(* IEC 61131-3 sources: ATCMcontrol_Engineering/src/TargetBase/Libs/ATCM_IEC1131_3/table_22, 158 files *)

(* ---- bool_to_byte.st ---- *)
(*[[
    UserURL= "ATCMfile:BOOL_TO_BYTE.htm"
]]*)

FUNCTION BOOL_TO_BYTE : BYTE
VAR_INPUT
    IN : BOOL;
END_VAR

inline { VMOP(bool_to_byte) }

END_FUNCTION

(* ---- bool_to_dint.st ---- *)
(*[[
    UserURL= "ATCMfile:BOOL_TO_DINT.htm"
]]*)

FUNCTION BOOL_TO_DINT : DINT
VAR_INPUT
    IN : BOOL;
END_VAR

inline{ VMOP(bool_to_dword) }

END_FUNCTION

(* ---- bool_to_dword.st ---- *)
(*[[
    UserURL= "ATCMfile:BOOL_TO_DWORD.htm"
]]*)

FUNCTION BOOL_TO_DWORD : DWORD
VAR_INPUT
    IN : BOOL;
END_VAR

inline{ VMOP(bool_to_dword) }

END_FUNCTION

(* ---- bool_to_int.st ---- *)
(*[[
    UserURL= "ATCMfile:BOOL_TO_DINT.htm"
]]*)

FUNCTION BOOL_TO_INT : INT
VAR_INPUT
    IN : BOOL;
END_VAR

inline{ VMOP(bool_to_word) }

END_FUNCTION

(* ---- bool_to_lreal.st ---- *)
(*[[
    UserURL= "ATCMfile:BOOL_TO_LREAL.htm"
]]*)

FUNCTION BOOL_TO_LREAL : LREAL
VAR_INPUT
    IN : BOOL;
END_VAR

inline{ VMOP(BOOL_TO_LREAL) }

END_FUNCTION

(* ---- bool_to_real.st ---- *)
(*[[
    UserURL= "ATCMfile:BOOL_TO_LREAL.htm"
]]*)

FUNCTION BOOL_TO_REAL : REAL
VAR_INPUT
    IN : BOOL;
END_VAR

inline{ VMOP }

END_FUNCTION

(* ---- bool_to_string.st ---- *)
(*[[
    UserURL= "ATCMfile:BOOL_TO_WSTRING.htm"
]]*)

FUNCTION BOOL_TO_STRING : STRING
VAR_INPUT
    IN : BOOL;
END_VAR

inline{ STDLIB(bool_to_string) }

END_FUNCTION

(* ---- bool_to_udint.st ---- *)
(*[[
    UserURL= "ATCMfile:BOOL_TO_UDINT.htm"
]]*)
FUNCTION BOOL_TO_UDINT : UDINT
VAR_INPUT
    IN : BOOL;
END_VAR

inline{ VMOP }

END_FUNCTION

(* ---- bool_to_uint.st ---- *)
(*[[
    UserURL= "ATCMfile:BOOL_TO_UINT.htm"
]]*)
FUNCTION BOOL_TO_UINT : UINT
VAR_INPUT
    IN : BOOL;
END_VAR

inline{ VMOP }

END_FUNCTION

(* ---- bool_to_word.st ---- *)
(*[[
    UserURL= "ATCMfile:BOOL_TO_WORD.htm"
]]*)

FUNCTION BOOL_TO_WORD : WORD
VAR_INPUT
    IN : BOOL;
END_VAR

inline{ VMOP }

END_FUNCTION

(* ---- byte_to_bool.st ---- *)
(*[[
    UserURL= "ATCMfile:BYTE_TO_BOOL.htm"
]]*)

FUNCTION BYTE_TO_BOOL : BOOL
VAR_INPUT
    IN : BYTE;
END_VAR

inline{VMOP}

END_FUNCTION

(* ---- byte_to_dint.st ---- *)
(*[[
    UserURL= "ATCMfile:BYTE_TO_DINT.htm"
]]*)

FUNCTION BYTE_TO_DINT : DINT
VAR_INPUT
    IN : BYTE;
END_VAR

inline{ VMOP(byte_to_dword) }

END_FUNCTION

(* ---- byte_to_dword.st ---- *)
(*[[
    UserURL= "ATCMfile:BYTE_TO_DWORD.htm"
]]*)

FUNCTION BYTE_TO_DWORD : DWORD
VAR_INPUT
    IN : BYTE;
END_VAR

inline{ VMOP }

END_FUNCTION

(* ---- byte_to_int.st ---- *)
(*[[
    UserURL= "ATCMfile:BYTE_TO_DINT.htm"
]]*)

FUNCTION BYTE_TO_INT : INT
VAR_INPUT
    IN : BYTE;
END_VAR

inline{ VMOP(byte_to_word) }

END_FUNCTION

(* ---- byte_to_lreal.st ---- *)
(*[[
    UserURL= "ATCMfile:BYTE_TO_LREAL.htm"
]]*)

FUNCTION BYTE_TO_LREAL : LREAL
VAR_INPUT
    IN : BYTE;
END_VAR

inline{VMOP}

END_FUNCTION

(* ---- byte_to_real.st ---- *)
(*[[
    UserURL= "ATCMfile:BYTE_TO_LREAL.htm"
]]*)

FUNCTION BYTE_TO_REAL : REAL
VAR_INPUT
    IN : BYTE;
END_VAR

inline{VMOP}

END_FUNCTION

(* ---- byte_to_string.st ---- *)
(*[[
    UserURL= "ATCMfile:BYTE_TO_WSTRING.htm"
]]*)

FUNCTION BYTE_TO_STRING : STRING
VAR_INPUT
    IN : BYTE;
END_VAR

inline{ STDLIB(byte_to_string) }

END_FUNCTION

(* ---- byte_to_udint.st ---- *)
(*[[
    UserURL= "ATCMfile:BYTE_TO_UDINT.htm"
]]*)
FUNCTION BYTE_TO_UDINT : UDINT
VAR_INPUT
    IN : BYTE;
END_VAR

inline{ VMOP }

END_FUNCTION

(* ---- byte_to_uint.st ---- *)
(*[[
    UserURL= "ATCMfile:BYTE_TO_UINT.htm"
]]*)
FUNCTION BYTE_TO_UINT : UINT
VAR_INPUT
    IN : BYTE;
END_VAR

inline{ VMOP }

END_FUNCTION

(* ---- byte_to_word.st ---- *)
(*[[
    UserURL= "ATCMfile:BYTE_TO_WORD.htm"
]]*)

FUNCTION BYTE_TO_WORD : WORD
VAR_INPUT
    IN : BYTE;
END_VAR

inline{VMOP}

END_FUNCTION

(* ---- dint_to_bool.st ---- *)
(*[[
    UserURL= "ATCMfile:DINT_TO_BOOL.htm"
]]*)

FUNCTION DINT_TO_BOOL : BOOL
VAR_INPUT
    IN : DINT;
END_VAR

inline{ VMOP(dword_to_bool) }

END_FUNCTION

(* ---- dint_to_byte.st ---- *)
(*[[
    UserURL= "ATCMfile:DINT_TO_BYTE.htm"
]]*)

FUNCTION DINT_TO_BYTE : BYTE
VAR_INPUT
    IN : DINT;
END_VAR

inline{ VMOP }

END_FUNCTION

(* ---- dint_to_dword.st ---- *)
(*[[
    UserURL= "ATCMfile:DINT_TO_DWORD.htm"
]]*)

FUNCTION DINT_TO_DWORD : DWORD
VAR_INPUT
    IN : DINT;
END_VAR

inline{NOOP}

END_FUNCTION

(* ---- dint_to_int.st ---- *)
(*[[
    UserURL= "ATCMfile:DINT_TO_LINT.htm"
]]*)

FUNCTION DINT_TO_INT : INT
VAR_INPUT
    IN : DINT;
END_VAR

inline{VMOP}

END_FUNCTION

(* ---- dint_to_lreal.st ---- *)
(*[[
    UserURL= "ATCMfile:DINT_TO_LREAL.htm"
]]*)

FUNCTION DINT_TO_LREAL : LREAL
VAR_INPUT
    IN : DINT;
END_VAR

inline{VMOP}

END_FUNCTION

(* ---- dint_to_real.st ---- *)
(*[[
    UserURL= "ATCMfile:DINT_TO_LREAL.htm"
]]*)

FUNCTION DINT_TO_REAL : REAL
VAR_INPUT
    IN : DINT;
END_VAR

inline{VMOP}

END_FUNCTION

(* ---- dint_to_string.st ---- *)
(*[[
    UserURL= "ATCMfile:DINT_TO_WSTRING.htm"
]]*)

FUNCTION DINT_TO_STRING : STRING
VAR_INPUT
    IN : DINT;
END_VAR

inline{ STDLIB(dint_to_string) }

END_FUNCTION

(* ---- dint_to_time.st ---- *)
(*[[
    UserURL= "ATCMfile:DINT_TO_TIME.htm"
]]*)

FUNCTION DINT_TO_TIME : TIME
VAR_INPUT
    IN : DINT;
END_VAR

inline { %1 }

END_FUNCTION

(* ---- dint_to_udint.st ---- *)
(*[[
    UserURL= "ATCMfile:DINT_TO_UDINT.htm"
]]*)
FUNCTION DINT_TO_UDINT : UDINT
VAR_INPUT
    IN : DINT;
END_VAR

inline{NOOP}

END_FUNCTION

(* ---- dint_to_uint.st ---- *)
(*[[
    UserURL= "ATCMfile:DINT_TO_UINT.htm"
]]*)
FUNCTION DINT_TO_UINT : UINT
VAR_INPUT
    IN : DINT;
END_VAR

inline{ VMOP }

END_FUNCTION

(* ---- dint_to_word.st ---- *)
(*[[
    UserURL= "ATCMfile:DINT_TO_WORD.htm"
]]*)

FUNCTION DINT_TO_WORD : WORD
VAR_INPUT
    IN : DINT;
END_VAR

inline{VMOP}

END_FUNCTION

(* ---- dword_to_bool.st ---- *)
(*[[
    UserURL= "ATCMfile:DWORD_TO_BOOL.htm"
]]*)

FUNCTION DWORD_TO_BOOL : BOOL
VAR_INPUT
    IN : DWORD;
END_VAR

inline{VMOP}

END_FUNCTION

(* ---- dword_to_byte.st ---- *)
(*[[
    UserURL= "ATCMfile:DWORD_TO_BYTE.htm"
]]*)

FUNCTION DWORD_TO_BYTE : BYTE
VAR_INPUT
    IN : DWORD;
END_VAR

inline{VMOP}

END_FUNCTION

(* ---- dword_to_dint.st ---- *)
(*[[
    UserURL= "ATCMfile:DWORD_TO_DINT.htm"
]]*)

FUNCTION DWORD_TO_DINT : DINT
VAR_INPUT
    IN : DWORD;
END_VAR

inline{VMOP}

END_FUNCTION

(* ---- dword_to_int.st ---- *)
(*[[
    UserURL= "ATCMfile:DWORD_TO_LINT.htm"
]]*)

FUNCTION DWORD_TO_INT : INT
VAR_INPUT
    IN : DWORD;
END_VAR

inline{VMOP}

END_FUNCTION

(* ---- dword_to_lreal.st ---- *)
(*[[
    UserURL= "ATCMfile:DWORD_TO_LREAL.htm"
]]*)

FUNCTION DWORD_TO_LREAL : LREAL
VAR_INPUT
    IN : DWORD;
END_VAR

inline{VMOP}

END_FUNCTION

(* ---- dword_to_lword.st ---- *)
(*[[
    UserURL= "ATCMfile:DWORD_TO_LWORD.htm"
]]*)

FUNCTION DWORD_TO_LWORD : LWORD
VAR_INPUT
    IN : DWORD;
END_VAR

inline{VMOP}

END_FUNCTION

(* ---- dword_to_real.st ---- *)
(*[[
    UserURL= "ATCMfile:DWORD_TO_LREAL.htm"
]]*)

FUNCTION DWORD_TO_REAL : REAL
VAR_INPUT
    IN : DWORD;
END_VAR

inline{VMOP}

END_FUNCTION

(* ---- dword_to_string.st ---- *)
(*[[
    UserURL= "ATCMfile:DWORD_TO_WSTRING.htm"
]]*)

FUNCTION DWORD_TO_STRING : STRING
VAR_INPUT
    IN : DWORD;
END_VAR

inline{ STDLIB(dword_to_string) }

END_FUNCTION

(* ---- dword_to_udint.st ---- *)
(*[[
    UserURL= "ATCMfile:DWORD_TO_UDINT.htm"
]]*)
FUNCTION DWORD_TO_UDINT : UDINT
VAR_INPUT
    IN : DWORD;
END_VAR

inline{NOOP}

END_FUNCTION

(* ---- dword_to_uint.st ---- *)
(*[[
    UserURL= "ATCMfile:DWORD_TO_UINT.htm"
]]*)
FUNCTION DWORD_TO_UINT : UINT
VAR_INPUT
    IN : DWORD;
END_VAR

inline{ VMOP }

END_FUNCTION

(* ---- dword_to_word.st ---- *)
(*[[
    UserURL= "ATCMfile:DWORD_TO_WORD.htm"
]]*)

FUNCTION DWORD_TO_WORD : WORD
VAR_INPUT
    IN : DWORD;
END_VAR

inline{VMOP(dword_to_uint)}

END_FUNCTION

(* ---- int_to_bool.st ---- *)
(*[[
    UserURL= "ATCMfile:DINT_TO_BOOL.htm"
]]*)

FUNCTION INT_TO_BOOL : BOOL
VAR_INPUT
    IN : INT;
END_VAR

inline{VMOP(WORD_TO_BOOL)}

END_FUNCTION

(* ---- int_to_byte.st ---- *)
(*[[
    UserURL= "ATCMfile:DINT_TO_BYTE.htm"
]]*)

FUNCTION INT_TO_BYTE : BYTE
VAR_INPUT
    IN : INT;
END_VAR

inline{VMOP(word_to_byte)}

END_FUNCTION

(* ---- int_to_dint.st ---- *)
(*[[
    UserURL= "ATCMfile:DINT_TO_LINT.htm"
]]*)

FUNCTION INT_TO_DINT : DINT
VAR_INPUT
    IN : INT;
END_VAR

inline{VMOP}

END_FUNCTION

(* ---- int_to_dword.st ---- *)
(*[[
    UserURL= "ATCMfile:DINT_TO_DWORD.htm"
]]*)

FUNCTION INT_TO_DWORD : DWORD
VAR_INPUT
    IN : INT;
END_VAR

inline{VMOP(int_to_dword)}

END_FUNCTION

(* ---- int_to_lint.st ---- *)
(*[[
    UserURL= "ATCMfile:DINT_TO_LINT.htm"
]]*)

FUNCTION INT_TO_LINT : LINT
VAR_INPUT
    IN : INT;
END_VAR

inline{VMOP}

END_FUNCTION

(* ---- int_to_lreal.st ---- *)
(*[[
    UserURL= "ATCMfile:DINT_TO_LREAL.htm"
]]*)

FUNCTION INT_TO_LREAL : LREAL
VAR_INPUT
    IN : INT;
END_VAR

inline{VMOP}

END_FUNCTION

(* ---- int_to_real.st ---- *)
(*[[
    UserURL= "ATCMfile:DINT_TO_LREAL.htm"
]]*)

FUNCTION INT_TO_REAL : REAL
VAR_INPUT
    IN : INT;
END_VAR

inline{VMOP}

END_FUNCTION

(* ---- int_to_string.st ---- *)
(*[[
    UserURL= "ATCMfile:DINT_TO_WSTRING.htm"
]]*)

FUNCTION INT_TO_STRING : STRING
VAR_INPUT
    IN : INT;
END_VAR

inline{ STDLIB(int_to_string) }

END_FUNCTION

(* ---- int_to_time.st ---- *)
(*[[
    UserURL= "ATCMfile:DINT_TO_TIME.htm"
]]*)

FUNCTION INT_TO_TIME : TIME
VAR_INPUT
    IN : INT;
END_VAR

inline
{
	%1
	int_to_dint
}

END_FUNCTION

(* ---- int_to_udint.st ---- *)
(*[[
    UserURL= "ATCMfile:INT_TO_UDINT.htm"
]]*)
FUNCTION INT_TO_UDINT : UDINT
VAR_INPUT
    IN : INT;
END_VAR

inline{ VMOP }

END_FUNCTION

(* ---- int_to_uint.st ---- *)
(*[[
    UserURL= "ATCMfile:INT_TO_UINT.htm"
]]*)
FUNCTION INT_TO_UINT : UINT
VAR_INPUT
    IN : INT;
END_VAR

inline{NOOP}

END_FUNCTION

(* ---- int_to_word.st ---- *)
(*[[
    UserURL= "ATCMfile:DINT_TO_WORD.htm"
]]*)

FUNCTION INT_TO_WORD : WORD
VAR_INPUT
    IN : INT;
END_VAR

inline{NOOP}

END_FUNCTION

(* ---- lint_to_bool.st ---- *)
(*[[
    UserURL= "ATCMfile:LINT_TO_BOOL.htm"
]]*)

FUNCTION LINT_TO_BOOL : BOOL
VAR_INPUT
    IN : LINT;
END_VAR

inline{%1==0l?false:true}

END_FUNCTION

(* ---- lint_to_byte.st ---- *)
(*[[
    UserURL= "ATCMfile:LINT_TO_BYTE.htm"
]]*)

FUNCTION LINT_TO_BYTE : BYTE
VAR_INPUT
    IN : LINT;
END_VAR

inline{(int)%1&0xff}

END_FUNCTION

(* ---- lint_to_dint.st ---- *)
(*[[
    UserURL= "ATCMfile:LINT_TO_DINT.htm"
]]*)

FUNCTION LINT_TO_DINT : DINT
VAR_INPUT
    IN : LINT;
END_VAR

inline{(int)%1}

END_FUNCTION

(* ---- lint_to_dword.st ---- *)
(*[[
    UserURL= "ATCMfile:LINT_TO_DWORD.htm"
]]*)

FUNCTION LINT_TO_DWORD : DWORD
VAR_INPUT
    IN : LINT;
END_VAR

inline{(int)%1}

END_FUNCTION

(* ---- lint_to_int.st ---- *)
(*[[
    UserURL= "ATCMfile:LINT_TO_DINT.htm"
]]*)

FUNCTION LINT_TO_INT : INT
VAR_INPUT
    IN : LINT;
END_VAR

inline{(int)%1}

END_FUNCTION

(* ---- lint_to_lreal.st ---- *)
(*[[
    UserURL= "ATCMfile:LINT_TO_LREAL.htm"
]]*)

FUNCTION LINT_TO_LREAL : LREAL
VAR_INPUT
    IN : LINT;
END_VAR

inline{(double)%1}

END_FUNCTION

(* ---- lint_to_lword.st ---- *)
(*[[
    UserURL= "ATCMfile:LINT_TO_LWORD.htm"
]]*)

FUNCTION LINT_TO_LWORD : LWORD
VAR_INPUT
    IN : LINT;
END_VAR

inline{%1}

END_FUNCTION

(* ---- lint_to_real.st ---- *)
(*[[
    UserURL= "ATCMfile:LINT_TO_LREAL.htm"
]]*)

FUNCTION LINT_TO_REAL : REAL
VAR_INPUT
    IN : LINT;
END_VAR

inline{(double)%1}

END_FUNCTION

(* ---- lint_to_string.st ---- *)
(*[[
    UserURL= "ATCMfile:LINT_TO_WSTRING.htm"
]]*)

FUNCTION LINT_TO_STRING : STRING
VAR_INPUT
    IN : LINT;
END_VAR

inline{java.lang.Long.toString(%1)}

END_FUNCTION

(* ---- lint_to_time.st ---- *)
(*[[
    UserURL= "ATCMfile:LINT_TO_TIME.htm"
]]*)

FUNCTION LINT_TO_TIME : TIME
VAR_INPUT
    IN : LINT;
END_VAR

inline{%1}

END_FUNCTION

(* ---- lint_to_word.st ---- *)
(*[[
    UserURL= "ATCMfile:LINT_TO_WORD.htm"
]]*)

FUNCTION LINT_TO_WORD : WORD
VAR_INPUT
    IN : LINT;
END_VAR

inline{(int)%1&0xffff}

END_FUNCTION

(* ---- lreal_to_bool.st ---- *)
(*[[
    UserURL= "ATCMfile:LREAL_TO_BOOL.htm"
]]*)

FUNCTION LREAL_TO_BOOL : BOOL
VAR_INPUT
    IN : LREAL;
END_VAR

inline{VMOP}

END_FUNCTION

(* ---- lreal_to_byte.st ---- *)
(*[[
    UserURL= "ATCMfile:LREAL_TO_BYTE.htm"
]]*)

FUNCTION LREAL_TO_BYTE : BYTE
VAR_INPUT
    IN : LREAL;
END_VAR

inline{VMOP}

END_FUNCTION

(* ---- lreal_to_dint.st ---- *)
(*[[
    UserURL= "ATCMfile:LREAL_TO_DINT.htm"
]]*)

FUNCTION LREAL_TO_DINT : DINT
VAR_INPUT
    IN : LREAL;
END_VAR

inline{VMOP}

END_FUNCTION

(* ---- lreal_to_dword.st ---- *)
(*[[
    UserURL= "ATCMfile:LREAL_TO_DWORD.htm"
]]*)

FUNCTION LREAL_TO_DWORD : DWORD
VAR_INPUT
    IN : LREAL;
END_VAR

inline{VMOP}

END_FUNCTION

(* ---- lreal_to_int.st ---- *)
(*[[
    UserURL= "ATCMfile:LREAL_TO_LINT.htm"
]]*)

FUNCTION LREAL_TO_INT : INT
VAR_INPUT
    IN : LREAL;
END_VAR

inline{VMOP}

END_FUNCTION

(* ---- lreal_to_lint.st ---- *)
(*[[
    UserURL= "ATCMfile:LREAL_TO_LINT.htm"
]]*)

FUNCTION LREAL_TO_LINT : LINT
VAR_INPUT
    IN : LREAL;
END_VAR

inline{VMOP(not_yet_implem)}

END_FUNCTION

(* ---- lreal_to_lword.st ---- *)
(*
 * Note:
 *  LREAL_TO_LWORD(x) is the same as
 *  LINT_TO_LWORD(LREAL_TO_LINT(x))
 *
 *  e.g.  LREAL_TO_LWORD(-1.0E0) = 16#ffffffffffffffff;
 *)

FUNCTION LREAL_TO_LWORD : LWORD
VAR_INPUT
    IN : LREAL;
END_VAR

inline{VMOP(not_yet_implem)}

END_FUNCTION

(* ---- lreal_to_real.st ---- *)
(*[[
    UserURL= "ATCMfile:LREAL_TO_TIME.htm"
]]*)

FUNCTION LREAL_TO_REAL : REAL
VAR_INPUT
    IN : LREAL;
END_VAR

inline{VMOP}

END_FUNCTION

(* ---- lreal_to_string.st ---- *)
(*[[
    UserURL= "ATCMfile:LREAL_TO_WSTRING.htm"
]]*)

FUNCTION LREAL_TO_STRING : STRING
VAR_INPUT
    IN : LREAL;
END_VAR

inline{ STDLIB(lreal_to_string)}

END_FUNCTION

(* ---- lreal_to_time.st ---- *)
(*[[
    UserURL= "ATCMfile:LREAL_TO_TIME.htm"
]]*)

FUNCTION LREAL_TO_TIME : TIME
VAR_INPUT
    IN : LREAL;
END_VAR

inline
{
    %1
	lreal_to_dint
}

END_FUNCTION

(* ---- lreal_to_udint.st ---- *)
(*[[
    UserURL= "ATCMfile:LREAL_TO_UDINT.htm"
]]*)
FUNCTION LREAL_TO_UDINT : UDINT
VAR_INPUT
    IN : LREAL;
END_VAR

inline{ VMOP }

END_FUNCTION

(* ---- lreal_to_uint.st ---- *)
(*[[
    UserURL= "ATCMfile:LREAL_TO_UINT.htm"
]]*)
FUNCTION LREAL_TO_UINT : UINT
VAR_INPUT
    IN : LREAL;
END_VAR

inline{ VMOP }

END_FUNCTION

(* ---- lreal_to_word.st ---- *)
(*[[
    UserURL= "ATCMfile:LREAL_TO_WORD.htm"
]]*)

FUNCTION LREAL_TO_WORD : WORD
VAR_INPUT
    IN : LREAL;
END_VAR

inline{VMOP}

END_FUNCTION

(* ---- lword_to_bool.st ---- *)
(*[[
    UserURL= "ATCMfile:LWORD_TO_BOOL.htm"
]]*)

FUNCTION LWORD_TO_BOOL : BOOL
VAR_INPUT
    IN : LWORD;
END_VAR

inline{%1==0l?false:true}

END_FUNCTION

(* ---- lword_to_byte.st ---- *)
(*[[
    UserURL= "ATCMfile:LWORD_TO_BYTE.htm"
]]*)

FUNCTION LWORD_TO_BYTE : BYTE
VAR_INPUT
    IN : LWORD;
END_VAR

inline{(int)%1&0xff}

END_FUNCTION

(* ---- lword_to_dint.st ---- *)
(*[[
    UserURL= "ATCMfile:LWORD_TO_DINT.htm"
]]*)

FUNCTION LWORD_TO_DINT : DINT
VAR_INPUT
    IN : LWORD;
END_VAR

inline{(int)%1}

END_FUNCTION

(* ---- lword_to_dword.st ---- *)
(*[[
    UserURL= "ATCMfile:LWORD_TO_DWORD.htm"
]]*)

FUNCTION LWORD_TO_DWORD : DWORD
VAR_INPUT
    IN : LWORD;
END_VAR

inline{(int)%1}

END_FUNCTION

(* ---- lword_to_int.st ---- *)
(*[[
    UserURL= "ATCMfile:LWORD_TO_DINT.htm"
]]*)

FUNCTION LWORD_TO_INT : INT
VAR_INPUT
    IN : LWORD;
END_VAR

inline{(int)%1}

END_FUNCTION

(* ---- lword_to_lint.st ---- *)
(*[[
    UserURL= "ATCMfile:LWORD_TO_LINT.htm"
]]*)

FUNCTION LWORD_TO_LINT : LINT
VAR_INPUT
    IN : LWORD;
END_VAR

inline{%1}

END_FUNCTION

(* ---- lword_to_lreal.st ---- *)
(*
 * Note:
 *  LWORD_TO_LREAL(x) is the same as
 *  LINT_TO_LREAL(LWORD_TO_LINT(x))
 *
 *  e.g.  LWORD_TO_LREAL(16#ffffffffffffffff) = -1.0E0
 *)
FUNCTION LWORD_TO_LREAL : LREAL
VAR_INPUT
    IN : LWORD;
END_VAR

inline{(double)%1}

END_FUNCTION

(* ---- lword_to_real.st ---- *)
(*
 * Note:
 *  LWORD_TO_LREAL(x) is the same as
 *  LINT_TO_LREAL(LWORD_TO_LINT(x))
 *
 *  e.g.  LWORD_TO_LREAL(16#ffffffffffffffff) = -1.0E0
 *)
FUNCTION LWORD_TO_REAL : REAL
VAR_INPUT
    IN : LWORD;
END_VAR

inline{(double)%1}

END_FUNCTION

(* ---- lword_to_string.st ---- *)
(*[[
    UserURL= "ATCMfile:LWORD_TO_WSTRING.htm"
]]*)

FUNCTION LWORD_TO_STRING : STRING
VAR_INPUT
    IN : LWORD;
END_VAR

inline{ STDLIB(not yet implemented) }

END_FUNCTION

(* ---- lword_to_word.st ---- *)
(*[[
    UserURL= "ATCMfile:LWORD_TO_WORD.htm"
]]*)

FUNCTION LWORD_TO_WORD : WORD
VAR_INPUT
    IN : LWORD;
END_VAR

inline{(int)%1&0xffff}

END_FUNCTION

(* ---- real_to_bool.st ---- *)
(*[[
    UserURL= "ATCMfile:REAL_TO_BOOL.htm"
]]*)

FUNCTION REAL_TO_BOOL : BOOL
VAR_INPUT
    IN : REAL;
END_VAR

inline{VMOP}

END_FUNCTION

(* ---- real_to_byte.st ---- *)
(*[[
    UserURL= "ATCMfile:REAL_TO_BYTE.htm"
]]*)

FUNCTION REAL_TO_BYTE : BYTE
VAR_INPUT
    IN : REAL;
END_VAR

inline{VMOP}

END_FUNCTION

(* ---- real_to_dint.st ---- *)
(*[[
    UserURL= "ATCMfile:REAL_TO_DINT.htm"
]]*)

FUNCTION REAL_TO_DINT : DINT
VAR_INPUT
    IN : REAL;
END_VAR

inline{VMOP}

END_FUNCTION

(* ---- real_to_dword.st ---- *)
(*[[
    UserURL= "ATCMfile:REAL_TO_DWORD.htm"
]]*)

FUNCTION REAL_TO_DWORD : DWORD
VAR_INPUT
    IN : REAL;
END_VAR

inline{VMOP}

END_FUNCTION

(* ---- real_to_int.st ---- *)
(*[[
    UserURL= "ATCMfile:REAL_TO_INT.htm"
]]*)

FUNCTION REAL_TO_INT : INT
VAR_INPUT
    IN : REAL;
END_VAR

inline{VMOP}

END_FUNCTION

(* ---- real_to_lint.st ---- *)
(*[[
    UserURL= "ATCMfile:REAL_TO_LINT.htm"
]]*)

FUNCTION REAL_TO_LINT : LINT
VAR_INPUT
    IN : REAL;
END_VAR

inline{VMOP(not_yet_implem)}

END_FUNCTION

(* ---- real_to_lreal.st ---- *)
(*[[
    UserURL= "ATCMfile:REAL_TO_LREAL.htm"
]]*)

FUNCTION REAL_TO_LREAL : LREAL
VAR_INPUT
    IN : REAL;
END_VAR

inline{VMOP}

END_FUNCTION

(* ---- real_to_lword.st ---- *)
(*[[
    UserURL= "ATCMfile:REAL_TO_LWORD.htm"
]]*)

FUNCTION REAL_TO_LWORD : LWORD
VAR_INPUT
    IN : REAL;
END_VAR

inline{VMOP(not_yet_implem)}

END_FUNCTION

(* ---- real_to_string.st ---- *)
(*[[
    UserURL= "ATCMfile:REAL_TO_STRING.htm"
]]*)

FUNCTION REAL_TO_STRING : STRING
VAR_INPUT
    IN : REAL;
END_VAR

inline{ STDLIB(real_to_string) }

END_FUNCTION

(* ---- real_to_time.st ---- *)
(*[[
    UserURL= "ATCMfile:REAL_TO_TIME.htm"
]]*)

FUNCTION REAL_TO_TIME : TIME
VAR_INPUT
    IN : REAL;
END_VAR

inline
{
    %1
    real_to_dint
}

END_FUNCTION

(* ---- real_to_udint.st ---- *)
(*[[
    UserURL= "ATCMfile:REAL_TO_UDINT.htm"
]]*)
FUNCTION REAL_TO_UDINT : UDINT
VAR_INPUT
    IN : REAL;
END_VAR

inline{ VMOP }

END_FUNCTION

(* ---- real_to_uint.st ---- *)
(*[[
    UserURL= "ATCMfile:REAL_TO_UINT.htm"
]]*)
FUNCTION REAL_TO_UINT : UINT
VAR_INPUT
    IN : REAL;
END_VAR

inline{ VMOP }

END_FUNCTION

(* ---- real_to_word.st ---- *)
(*[[
    UserURL= "ATCMfile:REAL_TO_WORD.htm"
]]*)

FUNCTION REAL_TO_WORD : WORD
VAR_INPUT
    IN : REAL;
END_VAR

inline{VMOP}

END_FUNCTION

(* ---- string_to_bool.st ---- *)
(*[[
    UserURL= "ATCMfile:WSTRING_TO_BOOL.htm"
]]*)

FUNCTION STRING_TO_BOOL : BOOL
VAR_INPUT
    IN : STRING;
END_VAR

inline { STDLIB(string_to_bool) }

END_FUNCTION

(* ---- string_to_byte.st ---- *)
(*[[
    UserURL= "ATCMfile:STRING_TO_BYTE.htm"
]]*)

FUNCTION STRING_TO_BYTE : BYTE
VAR_INPUT
    IN : STRING;
END_VAR

inline{ STDLIB(string_to_byte) }

END_FUNCTION

(* ---- string_to_date.st ---- *)
(*[[
    UserURL= "ATCMfile:STRING_TO_DATE.htm"
]]*)

FUNCTION STRING_TO_DATE : DATE
VAR_INPUT
    IN : STRING;
END_VAR

inline{ STDLIB(string_to_date) }

END_FUNCTION

(* ---- string_to_dint.st ---- *)
(*[[
    UserURL= "ATCMfile:WSTRING_TO_DINT.htm"
]]*)

FUNCTION STRING_TO_DINT : DINT
VAR_INPUT
    IN : STRING;
END_VAR

inline{ STDLIB(string_to_dint) }

END_FUNCTION

(* ---- string_to_dt.st ---- *)
(*[[
    UserURL= "ATCMfile:WSTRING_TO_DT.htm"
]]*)

FUNCTION STRING_TO_DT : DT
VAR_INPUT
    IN : STRING;
END_VAR

inline{VMOP(not_yet_implem)}

END_FUNCTION

(* ---- string_to_dword.st ---- *)
(*[[
    UserURL= "ATCMfile:WSTRING_TO_DWORD.htm"
]]*)

FUNCTION STRING_TO_DWORD : DWORD
VAR_INPUT
    IN : STRING;
END_VAR

inline{ STDLIB(string_to_dword) }

END_FUNCTION

(* ---- string_to_int.st ---- *)
(*[[
    UserURL= "ATCMfile:WSTRING_TO_LINT.htm"
]]*)

FUNCTION STRING_TO_INT : INT
VAR_INPUT
    IN : STRING;
END_VAR

inline{ STDLIB(string_to_int) }

END_FUNCTION

(* ---- string_to_lint.st ---- *)
(*[[
    UserURL= "ATCMfile:WSTRING_TO_LINT.htm"
]]*)

FUNCTION STRING_TO_LINT : LINT
VAR_INPUT
    IN : STRING;
END_VAR

inline{VMOP(not_yet_implem)}

END_FUNCTION

(* ---- string_to_lreal.st ---- *)
(*[[
    UserURL= "ATCMfile:WSTRING_TO_LREAL.htm"
]]*)

FUNCTION STRING_TO_LREAL : LREAL
VAR_INPUT
    IN : STRING;
END_VAR

inline{ STDLIB(string_to_lreal) }

END_FUNCTION

(* ---- string_to_lword.st ---- *)
(*[[
    UserURL= "ATCMfile:WSTRING_TO_LWORD.htm"
]]*)

FUNCTION STRING_TO_LWORD : LWORD
VAR_INPUT
    IN : STRING;
END_VAR

inline{VMOP(not_yet_implem)}

END_FUNCTION

(* ---- string_to_real.st ---- *)
(*[[
    UserURL= "ATCMfile:WSTRING_TO_LREAL.htm"
]]*)

FUNCTION STRING_TO_REAL : REAL
VAR_INPUT
    IN : STRING;
END_VAR

inline{ STDLIB(string_to_real) }
END_FUNCTION

(* ---- string_to_time.st ---- *)
(*[[
    UserURL= "ATCMfile:WSTRING_TO_TIME.htm"
]]*)

FUNCTION STRING_TO_TIME : TIME
VAR_INPUT
    IN : STRING;
END_VAR

inline{ STDLIB(string_to_time) }

END_FUNCTION

(* ---- string_to_tod.st ---- *)
(*[[
    UserURL= "ATCMfile:WSTRING_TO_TOD.htm"
]]*)

FUNCTION STRING_TO_TOD : TOD
VAR_INPUT
    IN : STRING;
END_VAR

inline{VMOP(not_yet_implem)}

END_FUNCTION

(* ---- string_to_udint.st ---- *)
(*[[
    UserURL= "ATCMfile:STRING_TO_UDINT.htm"
]]*)
FUNCTION STRING_TO_UDINT : UDINT
VAR_INPUT
    IN : STRING;
END_VAR

inline{ STDLIB(string_to_dword) }

END_FUNCTION

(* ---- string_to_uint.st ---- *)
(*[[
    UserURL= "ATCMfile:STRING_TO_UINT.htm"
]]*)
FUNCTION STRING_TO_UINT : UINT
VAR_INPUT
    IN : STRING;
END_VAR

inline{ STDLIB(string_to_word) }

END_FUNCTION

(* ---- string_to_word.st ---- *)
(*[[
    UserURL= "ATCMfile:WSTRING_TO_WORD.htm"
]]*)

FUNCTION STRING_TO_WORD : WORD
VAR_INPUT
    IN : STRING;
END_VAR

inline{ STDLIB(string_to_word) }

END_FUNCTION

(* ---- time_to_dint.st ---- *)
(*[[
    UserURL= "ATCMfile:TIME_TO_DINT.htm"
]]*)

FUNCTION TIME_TO_DINT : DINT
VAR_INPUT
    IN : TIME;
END_VAR

inline { %1 }

END_FUNCTION

(* ---- time_to_dt.st ---- *)
(*[[
    UserURL= "ATCMfile:TIME_TO_DT.htm"
]]*)

FUNCTION TIME_TO_DT : DT
VAR_INPUT
    IN : TIME;
END_VAR

inline{%1}

END_FUNCTION

(* ---- time_to_int.st ---- *)
(*[[
    UserURL= "ATCMfile:TIME_TO_LINT.htm"
]]*)

FUNCTION TIME_TO_INT : INT
VAR_INPUT
    IN : TIME;
END_VAR

inline
{
    %1
    dint_to_int
}

END_FUNCTION

(* ---- time_to_lint.st ---- *)
(*[[
    UserURL= "ATCMfile:TIME_TO_LINT.htm"
]]*)

FUNCTION TIME_TO_LINT : LINT
VAR_INPUT
    IN : TIME;
END_VAR

inline{%1}

END_FUNCTION

(* ---- time_to_lreal.st ---- *)
(*[[
    UserURL= "ATCMfile:TIME_TO_LREAL.htm"
]]*)

FUNCTION TIME_TO_LREAL : LREAL
VAR_INPUT
    IN : TIME;
END_VAR

inline
{
    %1
    dint_to_lreal
}

END_FUNCTION

(* ---- time_to_real.st ---- *)
(*[[
    UserURL= "ATCMfile:TIME_TO_LREAL.htm"
]]*)

FUNCTION TIME_TO_REAL : REAL
VAR_INPUT
    IN : TIME;
END_VAR

inline
{
    %1
    dint_to_real
}

END_FUNCTION

(* ---- time_to_string.st ---- *)
(*[[
    UserURL= "ATCMfile:TIME_TO_WSTRING.htm"
]]*)

FUNCTION TIME_TO_STRING : STRING
VAR_INPUT
   IN : TIME;
END_VAR

inline{ STDLIB(time32_to_string) }

END_FUNCTION

(* ---- tod_to_string.st ---- *)
(*[[
    UserURL= "ATCMfile:TOD_TO_STRING.htm"
]]*)

FUNCTION TOD_TO_STRING : STRING
VAR_INPUT
    IN : TOD;
END_VAR

inline{ STDLIB(not yet implented) }

END_FUNCTION

(* ---- tod_to_time.st ---- *)
(*[[
    UserURL= "ATCMfile:TOD_TO_TIME.htm"
]]*)

FUNCTION TOD_TO_TIME : TIME
VAR_INPUT
    IN : TOD;
END_VAR

inline{(long)%1}

END_FUNCTION

(* ---- trunc.st ---- *)
(*[[
    UserURL= "ATCMfile:TRUNC.htm"
]]*)

FUNCTION TRUNC : ANY_INT
VAR_INPUT
    IN : ANY_REAL;
END_VAR

overload DINT        (REAL)  inline{ STDLIB(Trunc_real_dint) }
overload DINT        (LREAL) inline{ STDLIB(Trunc_lreal_dint) }
overload DINT to INT (REAL)  inline{ STDLIB(Trunc_real_dint) }
overload DINT to INT (LREAL) inline{ STDLIB(Trunc_lreal_dint) }

END_FUNCTION

(* ---- udint_to_bool.st ---- *)
(*[[
    UserURL= "ATCMfile:UDINT_TO_BOOL.htm"
]]*)
FUNCTION UDINT_TO_BOOL : BOOL
VAR_INPUT
    IN : UDINT;
END_VAR

inline{ VMOP }

END_FUNCTION

(* ---- udint_to_byte.st ---- *)
(*[[
    UserURL= "ATCMfile:UDINT_TO_BYTE.htm"
]]*)
FUNCTION UDINT_TO_BYTE : BYTE
VAR_INPUT
    IN : UDINT;
END_VAR

inline{ VMOP }

END_FUNCTION

(* ---- udint_to_dint.st ---- *)
(*[[
    UserURL= "ATCMfile:UDINT_TO_DINT.htm"
]]*)
FUNCTION UDINT_TO_DINT : DINT
VAR_INPUT
    IN : UDINT;
END_VAR

inline{NOOP}

END_FUNCTION

(* ---- udint_to_dword.st ---- *)
(*[[
    UserURL= "ATCMfile:UDINT_TO_DWORD.htm"
]]*)
FUNCTION UDINT_TO_DWORD : DWORD
VAR_INPUT
    IN : UDINT;
END_VAR

inline{NOOP}

END_FUNCTION

(* ---- udint_to_int.st ---- *)
(*[[
    UserURL= "ATCMfile:UDINT_TO_INT.htm"
]]*)
FUNCTION UDINT_TO_INT : INT
VAR_INPUT
    IN : UDINT;
END_VAR

inline{ VMOP }

END_FUNCTION

(* ---- udint_to_lreal.st ---- *)
(*[[
    UserURL= "ATCMfile:UDINT_TO_LREAL.htm"
]]*)
FUNCTION UDINT_TO_LREAL : LREAL
VAR_INPUT
    IN : UDINT;
END_VAR

inline{ VMOP }

END_FUNCTION

(* ---- udint_to_real.st ---- *)
(*[[
    UserURL= "ATCMfile:UDINT_TO_REAL.htm"
]]*)
FUNCTION UDINT_TO_REAL : REAL
VAR_INPUT
    IN : UDINT;
END_VAR

inline{ VMOP }

END_FUNCTION

(* ---- udint_to_string.st ---- *)
(*[[
    UserURL= "ATCMfile:UDINT_TO_STRING.htm"
]]*)
FUNCTION UDINT_TO_STRING : STRING
VAR_INPUT
    IN : UDINT;
END_VAR

inline{ STDLIB(dword_to_string) }

END_FUNCTION

(* ---- udint_to_word.st ---- *)
(*[[
    UserURL= "ATCMfile:UDINT_TO_WORD.htm"
]]*)
FUNCTION UDINT_TO_WORD : WORD
VAR_INPUT
    IN : UDINT;
END_VAR

inline{ VMOP }

END_FUNCTION

(* ---- uint_to_bool.st ---- *)
(*[[
    UserURL= "ATCMfile:UINT_TO_BOOL.htm"
]]*)
FUNCTION UINT_TO_BOOL : BOOL
VAR_INPUT
    IN : UINT;
END_VAR

inline{ VMOP }

END_FUNCTION

(* ---- uint_to_byte.st ---- *)
(*[[
    UserURL= "ATCMfile:UINT_TO_BYTE.htm"
]]*)
FUNCTION UINT_TO_BYTE : BYTE
VAR_INPUT
    IN : UINT;
END_VAR

inline{ VMOP }

END_FUNCTION

(* ---- uint_to_dint.st ---- *)
(*[[
    UserURL= "ATCMfile:UINT_TO_DINT.htm"
]]*)
FUNCTION UINT_TO_DINT : DINT
VAR_INPUT
    IN : UINT;
END_VAR

inline{ VMOP }

END_FUNCTION

(* ---- uint_to_dword.st ---- *)
(*[[
    UserURL= "ATCMfile:UINT_TO_DWORD.htm"
]]*)
FUNCTION UINT_TO_DWORD : DWORD
VAR_INPUT
    IN : UINT;
END_VAR

inline{ VMOP }

END_FUNCTION

(* ---- uint_to_int.st ---- *)
(*[[
    UserURL= "ATCMfile:UINT_TO_INT.htm"
]]*)
FUNCTION UINT_TO_INT : INT
VAR_INPUT
    IN : UINT;
END_VAR

inline{NOOP}

END_FUNCTION

(* ---- uint_to_lreal.st ---- *)
(*[[
    UserURL= "ATCMfile:UINT_TO_LREAL.htm"
]]*)
FUNCTION UINT_TO_LREAL : LREAL
VAR_INPUT
    IN : UINT;
END_VAR

inline{ VMOP }

END_FUNCTION

(* ---- uint_to_real.st ---- *)
(*[[
    UserURL= "ATCMfile:UINT_TO_REAL.htm"
]]*)
FUNCTION UINT_TO_REAL : REAL
VAR_INPUT
    IN : UINT;
END_VAR

inline{ VMOP }

END_FUNCTION

(* ---- uint_to_string.st ---- *)
(*[[
    UserURL= "ATCMfile:UINT_TO_STRING.htm"
]]*)
FUNCTION UINT_TO_STRING : STRING
VAR_INPUT
    IN : UINT;
END_VAR

inline{ STDLIB(word_to_string) }

END_FUNCTION

(* ---- uint_to_word.st ---- *)
(*[[
    UserURL= "ATCMfile:UINT_TO_WORD.htm"
]]*)
FUNCTION UINT_TO_WORD : WORD
VAR_INPUT
    IN : UINT;
END_VAR

inline{NOOP}

END_FUNCTION

(* ---- word_string.st ---- *)
(*[[
    UserURL= "ATCMfile:WORD_TO_WSTRING.htm"
]]*)

FUNCTION WORD_TO_STRING : STRING
VAR_INPUT
    IN : WORD;
END_VAR

inline{VMOP}

END_FUNCTION

(* ---- word_to_bool.st ---- *)
(*[[
    UserURL= "ATCMfile:WORD_TO_BOOL.htm"
]]*)

FUNCTION WORD_TO_BOOL : BOOL
VAR_INPUT
    IN : WORD;
END_VAR

inline{VMOP}

END_FUNCTION

(* ---- word_to_byte.st ---- *)
(*[[
    UserURL= "ATCMfile:WORD_TO_BYTE.htm"
]]*)

FUNCTION WORD_TO_BYTE : BYTE
VAR_INPUT
    IN : WORD;
END_VAR

inline{VMOP}

END_FUNCTION

(* ---- word_to_dint.st ---- *)
(*[[
    UserURL= "ATCMfile:WORD_TO_DINT.htm"
]]*)

FUNCTION WORD_TO_DINT : DINT
VAR_INPUT
    IN : WORD;
END_VAR

inline{VMOP(word_to_dword)}

END_FUNCTION

(* ---- word_to_dword.st ---- *)
(*[[
    UserURL= "ATCMfile:WORD_TO_DWORD.htm"
]]*)

FUNCTION WORD_TO_DWORD : DWORD
VAR_INPUT
    IN : WORD;
END_VAR

inline{VMOP}

END_FUNCTION

(* ---- word_to_int.st ---- *)
(*[[
    UserURL= "ATCMfile:WORD_TO_INT.htm"
]]*)

FUNCTION WORD_TO_INT : INT
VAR_INPUT
    IN : WORD;
END_VAR

inline{NOOP}

END_FUNCTION

(* ---- word_to_lint.st ---- *)
(*[[
    UserURL= "ATCMfile:WORD_TO_LINT.htm"
]]*)

FUNCTION WORD_TO_LINT : LINT
VAR_INPUT
    IN : WORD;
END_VAR

inline{VMOP(not_yet_implem)}

END_FUNCTION

(* ---- word_to_lreal.st ---- *)
(*[[
    UserURL= "ATCMfile:WORD_TO_LREAL.htm"
]]*)

FUNCTION WORD_TO_LREAL : LREAL
VAR_INPUT
    IN : WORD;
END_VAR

inline{VMOP}

END_FUNCTION

(* ---- word_to_lword.st ---- *)
(*[[
    UserURL= "ATCMfile:WORD_TO_LWORD.htm"
]]*)

FUNCTION WORD_TO_LWORD : LWORD
VAR_INPUT
    IN : WORD;
END_VAR

inline{VMOP(not_yet_implem)}

END_FUNCTION

(* ---- word_to_real.st ---- *)
(*[[
    UserURL= "ATCMfile:WORD_TO_LREAL.htm"
]]*)

FUNCTION WORD_TO_REAL : REAL
VAR_INPUT
    IN : WORD;
END_VAR

inline{VMOP}

END_FUNCTION

(* ---- word_to_string.st ---- *)
(*[[
    UserURL= "ATCMfile:WORD_TO_WSTRING.htm"
]]*)

FUNCTION WORD_TO_STRING : STRING
VAR_INPUT
    IN : WORD;
END_VAR

inline{ STDLIB(word_to_string) }

END_FUNCTION

(* ---- word_to_udint.st ---- *)
(*[[
    UserURL= "ATCMfile:WORD_TO_UDINT.htm"
]]*)
FUNCTION WORD_TO_UDINT : UDINT
VAR_INPUT
    IN : WORD;
END_VAR

inline{ VMOP }

END_FUNCTION

(* ---- word_to_uint.st ---- *)
(*[[
    UserURL= "ATCMfile:WORD_TO_UINT.htm"
]]*)
FUNCTION WORD_TO_UINT : UINT
VAR_INPUT
    IN : WORD;
END_VAR

inline{NOOP}

END_FUNCTION
